Yaskawa INFORM job: X2_101(P)(125,-90)2.JBI

/JOB
//NAME X2_101(P)(125,-90)2
//POS
///NPOS 301,301,301,21,0,0
///TOOL 0
///POSTYPE PULSE
///PULSE
C00000=15474,202180,164610,0,0,38
C00001=2027,202198,164679,0,0,38
C00002=24736,215365,219614,34446,41710,-28276
C00003=32352,212431,219590,43411,47182,-30672
C00004=90146,188560,202920,30112,59119,-18336
C00005=118933,140461,218744,27304,53624,2807
C00006=105210,138110,229383,15554,54535,5056
C00007=120292,133807,224829,20615,58147,10246
C00008=120593,126537,218642,20775,58190,10295
C00009=120714,122004,214268,20769,58520,10378
C00010=120712,120035,212036,20692,58860,10445
C00011=120706,120595,212633,20705,58786,10429
C00012=120711,120851,214586,20937,57781,10229
C00013=120706,120595,212633,20705,58786,10429
C00014=120282,131035,221795,20517,58565,10327
C00015=120212,122631,223677,-19824,46644,-20033
C00016=120556,114962,216653,-19506,47024,-20076
C00017=120695,110312,211910,-19265,47534,-20168
C00018=120692,108202,209411,-19133,47963,-20258
C00019=120705,108724,209976,-19149,47889,-20241
C00020=120711,108700,211606,-19450,46928,-20036
C00021=120705,108724,209976,-19149,47889,-20241
C00022=120221,119783,220398,-19646,47168,-20147
C00023=120925,149751,244690,-34380,46703,-25518
C00024=121373,166523,227022,-36141,61926,-29055
C00025=120913,160748,223481,-36594,61174,-28897
C00026=120724,157112,220738,-36737,60983,-28874
C00027=120723,155199,218883,-36687,61111,-28923
C00028=120726,155677,219330,-36695,61088,-28913
C00029=120730,156730,222096,-37075,60150,-28553
C00030=120726,155677,219330,-36695,61088,-28913
C00031=121373,163920,224609,-36096,62046,-29099
C00032=120406,166637,227168,32311,57445,33728
C00033=120634,160817,223613,32676,56712,33541
C00034=120726,157198,220899,32780,56532,33504
C00035=120724,155250,219012,32723,56668,33550
C00036=120724,155690,219346,32716,56686,33555
C00037=120728,156742,222112,33132,55702,33215
C00038=120724,155690,219346,32716,56686,33555
C00039=120404,163997,224646,32246,57611,33783
C00040=133985,188744,240463,29202,55916,39414
C00041=133634,187862,227777,4842,42432,-77424
C00042=133983,183120,225880,4948,41153,-77374
C00043=134120,180360,224355,4989,40668,-77353
C00044=134108,178284,222610,4989,40676,-77358
C00045=134105,178637,222778,4981,40754,-77354
C00046=134286,180154,225906,5092,39605,-77360
C00047=134105,178637,222778,4981,40754,-77354
C00048=133615,185408,225690,4841,42456,-77429
C00049=121024,187697,227471,-25597,51015,-56291
C00050=120818,183050,225741,-26098,49773,-56012
C00051=120733,179873,223904,-26298,49302,-55905
C00052=120732,178247,222533,-26295,49309,-55908
C00053=120727,178630,222748,-26272,49366,-55926
C00054=120731,180176,225930,-26719,48320,-55616
C00055=120727,178630,222748,-26272,49366,-55926
C00056=121016,185268,225421,-25593,51025,-56296
C00057=120731,192327,238382,-525,21384,290
C00058=120720,184650,229554,-485,22872,268
C00059=120716,180491,225010,-470,23531,260
C00060=120714,178589,223412,-468,23537,258
C00061=120748,179412,224155,-490,23503,278
C00062=120744,177812,220907,-466,24679,265
C00063=120748,179412,224155,-490,23503,278
C00064=120764,190350,236905,-549,21277,311
C00065=148285,214402,237949,-4998,43525,10906
C00066=147844,206959,231028,-4889,43936,10712
C00067=147660,202909,227431,-4849,44060,10633
C00068=147643,201403,226399,-4857,43921,10635
C00069=147640,202124,226903,-4851,43981,10631
C00070=147319,200210,223567,-4711,45030,10450
C00071=147640,202124,226903,-4851,43981,10631
C00072=148254,212678,236902,-5015,43283,10908
C00073=144264,210294,243886,-8163,41086,13861
C00074=120755,180327,220298,-188,44229,164
C00075=120746,171881,211470,-184,45322,159
C00076=120742,168341,207661,-183,45847,157
C00077=120740,165439,205214,-182,45862,156
C00078=120719,166269,205935,-182,45844,148
C00079=120715,163797,201654,-178,47209,145
C00080=120719,166269,205935,-182,45844,148
C00081=120731,178408,218855,-188,44131,156
C00082=123087,177778,218562,-48004,45649,30777
C00083=121479,171146,210872,-47323,45938,29789
C00084=122530,166189,205678,-46713,46798,29742
C00085=122529,164979,204619,-46708,46819,29729
C00086=122529,165602,205165,-46719,46807,29736
C00087=122503,162924,200443,-45712,47877,29056
C00088=120838,166307,205861,-46999,46102,29364
C00089=120835,166361,205848,-46974,46126,29347
C00090=119861,166365,205849,-47111,45747,29113
C00091=120835,166361,205848,-46974,46126,29347
C00092=123074,175909,217070,-48037,45614,30794
C00093=121232,181774,235538,-27606,54021,27673
C00094=119095,158997,232657,-4189,63418,24156
C00095=116556,130755,220822,24696,63782,20050
C00096=116783,124225,216003,24912,63404,19994
C00097=116677,121428,213790,24861,63345,19966
C00098=124126,121440,213840,29408,62514,20795
C00099=124377,124183,215942,29533,62587,20852
C00100=123965,130725,220810,29194,62957,20896
C00101=125440,119589,219417,-31168,54029,-25826
C00102=124101,112544,213722,-32040,53801,-25914
C00103=124461,109637,211291,-31816,53838,-25883
C00104=115994,109663,211221,-37050,53005,-26653
C00105=116510,112581,213754,-36756,53014,-26588
C00106=116995,119639,219557,-36430,53113,-26564
C00107=126218,162099,239521,-28020,56999,-39411
C00108=123870,163328,223290,-28334,68014,-35019
C00109=122959,158598,221396,-29010,66719,-34890
C00110=123282,156546,220319,-28934,66438,-34739
C00111=117771,156561,220306,-31571,65347,-35721
C00112=117971,158636,221439,-31392,65705,-35782
C00113=118266,163418,223444,-30986,66822,-36040
C00114=120221,175834,229084,-3119,74575,4073
C00115=117582,163423,223451,27209,71262,31154
C00116=118328,158681,221539,27776,69997,31012
C00117=117739,156666,220543,27546,69730,30813
C00118=123312,156620,220547,30338,68636,31789
C00119=123482,158608,221419,30352,69024,31932
C00120=123188,163395,223433,29990,70147,32175
C00121=120067,178947,233192,25549,53044,55885
C00122=131070,185470,225867,7170,52227,-79323
C00123=131461,181907,225606,7389,50545,-79327
C00124=131646,180388,225354,7481,49912,-79321
C00125=136525,178881,222542,8029,50535,-77794
C00126=136445,180280,222598,7943,51220,-77765
C00127=135980,183829,222908,7713,52870,-77778
C00128=123522,184426,223985,-22802,61524,-57116
C00129=122967,181022,223967,-23325,59808,-56905
C00130=123040,179639,223960,-23465,59173,-56741
C00131=118101,179627,223904,-24803,58204,-57968
C00132=118290,181075,224034,-24590,58847,-58069
C00133=118546,184530,224142,-24121,60464,-58371
C00134=135828,184930,231784,3696,26075,2718
C00135=135741,176900,222633,3545,27580,2769
C00136=135898,173119,218034,3382,28468,2893
C00137=151866,161969,197943,-2562,35069,10366
C00138=151979,166024,202940,-2665,34080,10452
C00139=152363,175123,213641,-2941,32183,10704
C00140=121934,189549,236157,-2154,24440,9441
C00141=141176,183237,223578,-35123,36438,8037
C00142=140565,175008,214184,-33918,37549,7179
C00143=140340,171969,210603,-33443,38021,6842
C00144=125498,176939,219607,-33926,31237,2854
C00145=136257,146426,180013,-49389,59576,12695
C00146=136821,149913,184454,-49678,59198,13186
C00147=138256,158734,195155,-50257,58467,14304
C00148=90442,188267,218593,-20520,46484,-16259
C00149=38815,226894,234079,7619,30475,-17807
C00150=2027,202198,164679,0,0,38
C00151=15474,202180,164610,0,0,38
C00152=15474,202180,164610,0,0,38
C00153=15474,202180,164610,0,0,38
C00154=3643,-76224,-106676,19950,71810,76872
C00155=-17977,54134,16993,-10551,74333,28306
C00156=-37324,121541,115737,-14047,52289,7724
C00157=-48165,192898,197715,-15732,40765,-3970
C00158=-58614,195716,224396,-17895,28031,-14924
C00159=-138322,143321,229105,-42804,47301,-20408
C00160=-140817,146158,237227,-45779,45351,-19330
C00161=-147159,125749,218226,-45329,49662,-21330
C00162=-147437,121228,213779,-45242,49912,-21531
C00163=-147412,119200,211479,-45009,50185,-21684
C00164=-147407,119721,212016,-45043,50140,-21657
C00165=-147931,119949,213841,-45946,49334,-21289
C00166=-147407,119721,212016,-45043,50140,-21657
C00167=-146392,130285,221614,-44743,49966,-21354
C00168=-146532,144143,225646,4227,57465,17778
C00169=-147178,137204,219990,3902,57394,17672
C00170=-147427,133024,216151,3767,57613,17639
C00171=-147404,130928,213882,3765,57930,17654
C00172=-147409,131440,214347,3763,57908,17652
C00173=-147876,131929,216457,3567,56871,17542
C00174=-147409,131440,214347,3763,57908,17652
C00175=-146502,154568,235407,4272,56817,17758
C00176=-99845,140323,234668,41114,43975,29200
C00177=-130588,156406,235029,35449,55402,24493
C00178=-147611,165369,225951,24300,67303,24402
C00179=-147499,159686,222616,24499,66491,24247
C00180=-147440,155964,219836,24563,66297,24218
C00181=-147421,154162,218086,24545,66432,24252
C00182=-147416,154709,218664,24561,66363,24237
C00183=-147807,155692,221265,24569,65426,23941
C00184=-147416,154709,218664,24561,66363,24237
C00185=-147574,162825,223650,24300,67397,24430
C00186=-120351,165667,226538,-30553,61026,-29699
C00187=-120572,159826,222941,-30869,60298,-29533
C00188=-120662,156191,220198,-30959,60125,-29502
C00189=-120661,154235,218293,-30911,60269,-29546
C00190=-120662,154654,218578,-30900,60303,-29557
C00191=-120660,155573,221272,-31248,59284,-29233
C00192=-120662,154654,218578,-30900,60303,-29557
C00193=-120351,162993,223944,-30493,61219,-29757
C00194=-106019,170897,239329,-29591,39413,-48114
C00195=-120349,165701,226589,-30025,41462,-53269
C00196=-120571,159856,222988,-30524,40733,-53054
C00197=-120660,156245,220264,-30650,40558,-53013
C00198=-120659,154264,218337,-30550,40705,-53072
C00199=-120657,154705,218714,-30553,40700,-53069
C00200=-120657,155527,221042,-31160,39828,-52703
C00201=-120657,154705,218714,-30553,40700,-53069
C00202=-120346,163050,224086,-29924,41618,-53328
C00203=-121003,165681,226549,30422,41392,53375
C00204=-120764,159836,222944,30930,40664,53161
C00205=-120666,156628,220610,31078,40460,53111
C00206=-120665,154243,218290,30958,40635,53182
C00207=-120651,154718,218742,30981,40602,53173
C00208=-120645,155770,221512,31697,39599,52755
C00209=-120651,154718,218742,30981,40602,53173
C00210=-120988,163064,224120,30339,41520,53430
C00211=-145273,180969,224600,13907,25635,-13338
C00212=-150975,169052,202561,-14336,33678,-6171
C00213=-152120,157871,187736,-12805,36812,-7299
C00214=-151822,150501,178835,-12433,38503,-7437
C00215=-151822,147953,176273,-12361,38765,-7478
C00216=-151822,149084,177415,-12394,38645,-7460
C00217=-151589,146591,173415,-12167,39831,-7535
C00218=-151919,152197,181098,-12541,37982,-7398
C00219=-152280,169114,198720,-13043,35835,-7206
C00220=-158898,171274,210982,-44327,26584,1788
C00221=-158473,166641,205336,-42970,27544,1214
C00222=-157744,151580,188391,-39934,29853,-149
C00223=-157744,148965,185817,-39669,30040,-287
C00224=-157744,150293,187130,-39808,29943,-216
C00225=-157372,147876,183051,-38565,31072,-770
C00226=-157636,151887,188203,-39669,30105,-261
C00227=-158813,181767,219065,-43782,26920,1533
C00228=-129261,210513,245515,5534,45622,-8457
C00229=-125085,198862,239535,25777,46081,-13421
C00230=-119299,188173,224850,24885,48032,-10780
C00231=-120885,182304,217176,24168,49943,-10840
C00232=-120885,180234,215583,24199,49865,-10857
C00233=-120885,180747,215981,24191,49883,-10853
C00234=-120884,178818,212615,23832,50874,-10599
C00235=-120886,180612,215743,24164,49954,-10836
C00236=-120886,189219,222159,24004,50389,-10723
C00237=-108287,189347,219965,24064,48852,-6477
C00238=-108287,184786,216642,24169,48578,-6550
C00239=-108287,180112,213087,24246,48382,-6602
C00240=-108287,177544,211068,24278,48311,-6618
C00241=-108287,178306,211671,24271,48329,-6612
C00242=-108405,176503,208569,23922,49256,-6410
C00243=-108249,178868,212644,24384,48037,-6676
C00244=-121452,188951,222489,24083,50199,-10971
C00245=-121452,188951,222489,24083,50199,-10971
C00246=-122116,184054,218869,24132,50081,-11240
C00247=-122262,178348,212240,23732,51169,-11010
C00248=-108771,176193,208579,23747,49083,-6567
C00249=-111092,174695,211589,36295,46390,-11684
C00250=-112169,180872,218864,36952,45675,-12470
C00251=-113202,195859,242327,41337,40702,-15530
C00252=-130749,165712,222917,10388,27694,-8279
C00253=-152425,178401,240789,-26989,10054,1286
C00254=-149111,168631,221120,-26779,26556,407
C00255=-148536,165202,217049,-26272,27343,326
C00256=-159853,153774,193335,-13592,36205,-8842
C00257=-158113,149758,193299,-37101,31198,-1306
C00258=-158618,158017,203094,-38867,29614,-530
C00259=-160401,183295,230590,-43445,26035,1284
C00260=-117887,183372,223265,-22549,61468,-57164
C00261=-118052,179927,223173,-22955,59851,-56864
C00262=-118699,178546,222858,-23249,59248,-56921
C00263=-123672,178493,222758,-24591,58283,-58163
C00264=-123113,179961,223261,-24333,58805,-58120
C00265=-122866,183435,223403,-23872,60412,-58418
C00266=-123473,183399,223341,22943,61343,57288
C00267=-123290,179951,223242,23362,59727,56988
C00268=-123487,178672,223340,23471,59103,56791
C00269=-118424,178788,223621,24887,57983,58016
C00270=-118228,179938,223194,24724,58720,58254
C00271=-118494,183412,223341,24252,60324,58552
C00272=-131011,176479,228164,31225,71276,43628
C00273=-123827,162412,222773,27424,71320,31095
C00274=-123627,157628,220768,27711,70190,30861
C00275=-124009,155619,219621,27570,69971,30722
C00276=-118332,155649,219817,30457,68786,31689
C00277=-117906,157627,220734,30586,69092,31875
C00278=-118212,162433,222788,30219,70202,32114
C00279=-117529,162374,222654,-26899,71438,-31030
C00280=-117708,157592,220653,-27171,70307,-30797
C00281=-118564,155615,219745,-27674,69741,-30848
C00282=-124047,155559,219614,-30429,68730,-31821
C00283=-123427,157610,220727,-30053,69177,-31802
C00284=-123142,162415,222776,-29701,70290,-32041
C00285=-132073,148583,237547,-34621,60846,-21391
C00286=-129975,141241,222454,-31403,66136,-22661
C00287=-130468,135202,218431,-31833,65522,-22562
C00288=-131729,132640,216434,-32594,65253,-22701
C00289=-138385,131644,213865,-36199,65039,-23836
C00290=-137184,134500,216293,-35511,65228,-23678
C00291=-136557,140559,220416,-35003,65813,-23762
C00292=-150189,140118,219078,9123,71574,17400
C00293=-150541,134122,215115,8948,70956,17299
C00294=-151485,131353,212608,8387,71119,17166
C00295=-145176,132679,216974,12237,68813,17910
C00296=-144130,135523,219427,12862,68701,18051
C00297=-143910,141531,223338,12937,69351,18155
C00298=-134795,161184,236321,9699,64146,14551
C00299=-58614,195716,224396,-17895,28031,-14924
C00300=15474,202180,164610,0,0,38
BC00000=0,675528,1075229
BC00001=0,1249520,1075229
BC00002=20074,1273230,1075229
BC00003=22843,1276500,1075229
BC00004=181219,1349640,881743
BC00005=259614,1271622,997019
BC00006=263455,1253369,961473
BC00007=299365,1262893,899090
BC00008=299365,1262893,899090
BC00009=299365,1262893,899090
BC00010=299365,1262893,899090
BC00011=299365,1262893,899090
BC00012=299365,1262893,899090
BC00013=299365,1262893,899090
BC00014=299365,1262893,899090
BC00015=317385,1250080,966851
BC00016=317385,1250080,966851
BC00017=317385,1250080,966851
BC00018=317385,1250080,966851
BC00019=317385,1250080,966851
BC00020=317385,1250080,966851
BC00021=317385,1250080,966851
BC00022=317385,1250080,966851
BC00023=333821,1266832,919202
BC00024=286205,1304114,811613
BC00025=286205,1304114,811613
BC00026=286205,1304114,811613
BC00027=286205,1304114,811613
BC00028=286205,1304114,811613
BC00029=286205,1304114,811613
BC00030=286205,1304114,811613
BC00031=286205,1304114,811613
BC00032=312946,1307861,830398
BC00033=312946,1307861,830398
BC00034=312946,1307861,830398
BC00035=312946,1307861,830398
BC00036=312946,1307861,830398
BC00037=312946,1307861,830398
BC00038=312946,1307861,830398
BC00039=312946,1307861,830398
BC00040=309388,1296619,799441
BC00041=318547,1318060,813250
BC00042=318547,1318060,813250
BC00043=318547,1318060,813250
BC00044=318547,1318060,813250
BC00045=318547,1318060,813250
BC00046=318547,1318060,813250
BC00047=318547,1318060,813250
BC00048=318547,1318060,813250
BC00049=305027,1313604,795360
BC00050=305027,1313604,795360
BC00051=305027,1313604,795360
BC00052=305027,1313604,795360
BC00053=305027,1313604,795360
BC00054=305027,1313604,795360
BC00055=305027,1313604,795360
BC00056=305027,1313604,795360
BC00057=324377,1352422,788984
BC00058=324377,1352422,788984
BC00059=324377,1352422,788984
BC00060=324377,1352422,788984
BC00061=324377,1352422,788984
BC00062=324377,1352422,788984
BC00063=324377,1352422,788984
BC00064=324377,1352422,788984
BC00065=364692,1338716,661668
BC00066=364692,1338716,661668
BC00067=364692,1338716,661668
BC00068=364692,1338716,661668
BC00069=364692,1338716,661668
BC00070=364692,1338716,661668
BC00071=364692,1338716,661668
BC00072=364692,1338716,661668
BC00073=369598,1321086,746352
BC00074=329275,1315048,881081
BC00075=329275,1315048,881081
BC00076=329275,1315048,881081
BC00077=329275,1315048,881081
BC00078=329275,1315048,881081
BC00079=329275,1315048,881081
BC00080=329275,1315048,881081
BC00081=329275,1315048,881081
BC00082=314852,1330108,807446
BC00083=314852,1330108,807446
BC00084=314853,1330108,807444
BC00085=314853,1330108,807443
BC00086=314853,1330108,807443
BC00087=314853,1330108,807443
BC00088=314852,1330108,807446
BC00089=314852,1330108,807446
BC00090=314852,1330108,807446
BC00091=314852,1330108,807446
BC00092=314852,1330108,807446
BC00093=313257,1310637,824311
BC00094=311421,1288215,843732
BC00095=309154,1260535,867707
BC00096=309154,1260535,867707
BC00097=309154,1260535,867707
BC00098=309154,1260535,867707
BC00099=309154,1260535,867707
BC00100=309154,1260535,867707
BC00101=294407,1249819,928832
BC00102=294407,1249819,928832
BC00103=294407,1249819,928832
BC00104=294407,1249819,928832
BC00105=294407,1249819,928832
BC00106=294407,1249819,928832
BC00107=314801,1292959,892910
BC00108=293885,1292722,795471
BC00109=293885,1292722,795471
BC00110=293885,1292722,795471
BC00111=293885,1292722,795471
BC00112=293885,1292722,795471
BC00113=293885,1292722,795471
BC00114=299435,1291649,781795
BC00115=313202,1288383,786633
BC00116=313202,1288383,786633
BC00117=313202,1288383,786633
BC00118=313201,1288384,786631
BC00119=313202,1288383,786633
BC00120=313202,1288383,786633
BC00121=311248,1293583,920117
BC00122=320223,1301498,798955
BC00123=320223,1301498,798955
BC00124=320223,1301498,798955
BC00125=320223,1301498,798955
BC00126=320223,1301498,798955
BC00127=320223,1301498,798955
BC00128=303809,1297500,774731
BC00129=303809,1297500,774731
BC00130=303809,1297500,774731
BC00131=303809,1297500,774731
BC00132=303809,1297500,774731
BC00133=303809,1297500,774731
BC00134=382985,1337291,817528
BC00135=382985,1337291,817528
BC00136=382985,1337291,817528
BC00137=382985,1337291,817528
BC00138=382985,1337291,817528
BC00139=382985,1337291,817528
BC00140=326395,1340304,844891
BC00141=362940,1334773,820893
BC00142=362940,1334773,820893
BC00143=362940,1334773,820893
BC00144=362940,1334773,820893
BC00145=362940,1334773,820893
BC00146=362940,1334773,820893
BC00147=362940,1334773,820893
BC00148=199115,1355011,996382
BC00149=79950,1309724,1030230
BC00150=0,1249520,1075229
BC00151=0,675528,1075229
BC00152=0,675528,1075229
BC00153=0,675528,1075229
BC00154=199464,674570,1075173
BC00155=168150,723863,951549
BC00156=154085,663617,1001676
BC00157=146204,714236,1057448
BC00158=138607,763027,1056836
BC00159=343461,851890,923082
BC00160=347349,853577,920544
BC00161=364317,860937,909465
BC00162=364317,860937,909465
BC00163=364317,860937,909465
BC00164=364317,860937,909465
BC00165=364317,860937,909465
BC00166=364317,860937,909465
BC00167=364317,860937,909465
BC00168=379202,846237,874129
BC00169=379202,846237,874129
BC00170=379202,846237,874129
BC00171=379202,846237,874129
BC00172=379202,846237,874129
BC00173=379202,846237,874129
BC00174=379202,846237,874129
BC00175=379202,846237,874129
BC00176=267497,855485,958441
BC00177=320924,819371,961652
BC00178=359813,832026,812779
BC00179=359813,832026,812779
BC00180=359813,832026,812779
BC00181=359813,832026,812779
BC00182=359813,832026,812779
BC00183=359813,832026,812779
BC00184=359813,832026,812779
BC00185=359813,832026,812779
BC00186=313650,822927,822655
BC00187=313650,822927,822655
BC00188=313650,822927,822655
BC00189=313650,822927,822655
BC00190=313650,822927,822655
BC00191=313650,822927,822655
BC00192=313650,822927,822655
BC00193=313650,822927,822655
BC00194=268540,837164,928608
BC00195=303309,837622,929453
BC00196=303309,837622,929453
BC00197=303309,837622,929453
BC00198=303309,837622,929453
BC00199=303309,837622,929453
BC00200=303309,837622,929453
BC00201=303309,837622,929453
BC00202=303309,837622,929453
BC00203=306476,837214,930249
BC00204=306476,837214,930249
BC00205=306476,837214,930249
BC00206=306476,837214,930249
BC00207=306476,837214,930249
BC00208=306476,837214,930249
BC00209=306476,837214,930249
BC00210=306476,837214,930249
BC00211=398174,775712,811563
BC00212=398174,775712,811563
BC00213=398174,775712,811563
BC00214=398174,775712,811563
BC00215=398174,775712,811563
BC00216=398174,775712,811563
BC00217=398174,775712,811563
BC00218=398174,775712,811563
BC00219=398174,775712,811563
BC00220=398174,793888,811563
BC00221=398174,793888,811563
BC00222=398174,793888,811563
BC00223=398174,793888,811563
BC00224=398174,793888,811563
BC00225=398174,793888,811563
BC00226=398174,793888,811563
BC00227=398174,793888,811563
BC00228=296475,807012,791430
BC00229=296475,807012,791430
BC00230=296475,807012,791430
BC00231=296475,807012,791430
BC00232=296475,807012,791430
BC00233=296475,807012,791430
BC00234=296475,807012,791430
BC00235=296475,807012,791430
BC00236=296475,807012,791430
BC00237=296475,807012,791430
BC00238=296475,807012,791430
BC00239=296475,807012,791430
BC00240=296475,807012,791430
BC00241=296475,807012,791430
BC00242=296475,807012,791430
BC00243=296475,807012,791430
BC00244=296475,807012,791430
BC00245=296475,807012,791430
BC00246=296475,807012,791430
BC00247=296476,807010,791427
BC00248=296786,806946,791584
BC00249=296786,806946,791584
BC00250=296786,806946,791584
BC00251=296786,806946,791584
BC00252=343473,807454,949850
BC00253=383324,814067,855911
BC00254=383324,814067,855911
BC00255=383324,814067,855911
BC00256=383324,814066,855908
BC00257=383324,814067,855911
BC00258=383324,814067,855911
BC00259=383324,814067,855911
BC00260=304526,826961,775443
BC00261=304526,826961,775443
BC00262=304526,826961,775443
BC00263=304526,826961,775443
BC00264=304526,826961,775443
BC00265=304526,826961,775443
BC00266=305115,826537,776504
BC00267=305115,826537,776504
BC00268=305115,826537,776504
BC00269=305115,826537,776504
BC00270=305115,826537,776504
BC00271=305115,826537,776504
BC00272=317689,831131,771467
BC00273=295274,836215,786981
BC00274=295274,836215,786981
BC00275=295274,836215,786981
BC00276=295274,836215,786981
BC00277=295274,836215,786981
BC00278=295274,836215,786981
BC00279=313970,836931,785826
BC00280=313970,836931,785826
BC00281=313970,836931,785826
BC00282=313970,836931,785826
BC00283=313970,836931,785826
BC00284=313970,836931,785826
BC00285=304168,872987,860177
BC00286=340834,848874,817062
BC00287=340834,848874,817062
BC00288=340834,848874,817062
BC00289=340834,848874,817062
BC00290=340834,848874,817062
BC00291=340834,848874,817062
BC00292=360407,856018,818040
BC00293=360407,856018,818040
BC00294=360407,856018,818040
BC00295=360407,856018,818040
BC00296=360407,856018,818040
BC00297=360407,856018,818040
BC00298=336693,846075,843572
BC00299=138607,763027,1056836
BC00300=0,675528,1075229
EC00000=1108551,-556475
EC00001=1108551,-556475
EC00002=1108551,-556475
EC00003=1108551,-556475
EC00004=1108551,-556475
EC00005=1108551,-556475
EC00006=1108551,-556475
EC00007=1108551,-556475
EC00008=1108551,-556475
EC00009=1108551,-556475
EC00010=1108551,-556475
EC00011=1108551,-556475
EC00012=1108551,-556475
EC00013=1108551,-556475
EC00014=1108551,-556475
EC00015=1108551,-556475
EC00016=1108551,-556475
EC00017=1108551,-556475
EC00018=1108551,-556475
EC00019=1108551,-556475
EC00020=1108551,-556475
EC00021=1108551,-556475
EC00022=1108551,-556475
EC00023=1108551,-556475
EC00024=1108551,-556475
EC00025=1108551,-556475
EC00026=1108551,-556475
EC00027=1108551,-556475
EC00028=1108551,-556475
EC00029=1108551,-556475
EC00030=1108551,-556475
EC00031=1108551,-556475
EC00032=1108551,-556475
EC00033=1108551,-556475
EC00034=1108551,-556475
EC00035=1108551,-556475
EC00036=1108551,-556475
EC00037=1108551,-556475
EC00038=1108551,-556475
EC00039=1108551,-556475
EC00040=1108551,-556475
EC00041=1108551,-556475
EC00042=1108551,-556475
EC00043=1108551,-556475
EC00044=1108551,-556475
EC00045=1108551,-556475
EC00046=1108551,-556475
EC00047=1108551,-556475
EC00048=1108551,-556475
EC00049=1108551,-556475
EC00050=1108551,-556475
EC00051=1108551,-556475
EC00052=1108551,-556475
EC00053=1108551,-556475
EC00054=1108551,-556475
EC00055=1108551,-556475
EC00056=1108551,-556475
EC00057=1108551,-556475
EC00058=1108551,-556475
EC00059=1108551,-556475
EC00060=1108551,-556475
EC00061=1108551,-556475
EC00062=1108551,-556475
EC00063=1108551,-556475
EC00064=1108551,-556475
EC00065=1108551,-556475
EC00066=1108551,-556475
EC00067=1108551,-556475
EC00068=1108551,-556475
EC00069=1108551,-556475
EC00070=1108551,-556475
EC00071=1108551,-556475
EC00072=1108551,-556475
EC00073=1108551,-556475
EC00074=1108551,-556475
EC00075=1108551,-556475
EC00076=1108551,-556475
EC00077=1108551,-556475
EC00078=1108551,-556475
EC00079=1108551,-556475
EC00080=1108551,-556475
EC00081=1108551,-556475
EC00082=1108551,-556475
EC00083=1108551,-556475
EC00084=1108551,-556475
EC00085=1108550,-556475
EC00086=1108550,-556475
EC00087=1108550,-556475
EC00088=1108551,-556475
EC00089=1108551,-556475
EC00090=1108551,-556475
EC00091=1108551,-556475
EC00092=1108551,-556475
EC00093=1108551,-556475
EC00094=1108551,-556475
EC00095=1108551,-556475
EC00096=1108551,-556475
EC00097=1108551,-556475
EC00098=1108551,-556475
EC00099=1108551,-556475
EC00100=1108551,-556475
EC00101=1108551,-556475
EC00102=1108551,-556475
EC00103=1108551,-556475
EC00104=1108551,-556475
EC00105=1108551,-556475
EC00106=1108551,-556475
EC00107=1108551,-556475
EC00108=1108551,-556475
EC00109=1108551,-556475
EC00110=1108551,-556475
EC00111=1108551,-556475
EC00112=1108551,-556475
EC00113=1108551,-556475
EC00114=1108551,-556475
EC00115=1108551,-556475
EC00116=1108551,-556475
EC00117=1108551,-556475
EC00118=1108550,-556474
EC00119=1108551,-556475
EC00120=1108551,-556475
EC00121=1108551,-556475
EC00122=1108551,-556475
EC00123=1108551,-556475
EC00124=1108551,-556475
EC00125=1108551,-556475
EC00126=1108551,-556475
EC00127=1108551,-556475
EC00128=1108551,-556475
EC00129=1108551,-556475
EC00130=1108551,-556475
EC00131=1108551,-556475
EC00132=1108551,-556475
EC00133=1108551,-556475
EC00134=1108551,-556475
EC00135=1108551,-556475
EC00136=1108551,-556475
EC00137=1108551,-556475
EC00138=1108551,-556475
EC00139=1108551,-556475
EC00140=1108551,-556475
EC00141=1108551,-556475
EC00142=1108551,-556475
EC00143=1108551,-556475
EC00144=1108551,-556475
EC00145=1108551,-556475
EC00146=1108551,-556475
EC00147=1108551,-556475
EC00148=1108551,-556475
EC00149=1108551,-556475
EC00150=1108551,-556475
EC00151=1108551,-556475
EC00152=266052,-556475
EC00153=-266052,556475
EC00154=-1108551,556475
EC00155=-1108551,556475
EC00156=-1108551,556475
EC00157=-1108551,556475
EC00158=-1108551,556475
EC00159=-1108551,556475
EC00160=-1108551,556475
EC00161=-1108551,556475
EC00162=-1108551,556475
EC00163=-1108551,556475
EC00164=-1108551,556475
EC00165=-1108551,556475
EC00166=-1108551,556475
EC00167=-1108551,556475
EC00168=-1108551,556475
EC00169=-1108551,556475
EC00170=-1108551,556475
EC00171=-1108551,556475
EC00172=-1108551,556475
EC00173=-1108551,556475
EC00174=-1108551,556475
EC00175=-1108551,556475
EC00176=-1108551,556475
EC00177=-1108551,556475
EC00178=-1108551,556475
EC00179=-1108551,556475
EC00180=-1108551,556475
EC00181=-1108551,556475
EC00182=-1108551,556475
EC00183=-1108551,556475
EC00184=-1108551,556475
EC00185=-1108551,556475
EC00186=-1108551,556475
EC00187=-1108551,556475
EC00188=-1108551,556475
EC00189=-1108551,556475
EC00190=-1108551,556475
EC00191=-1108551,556475
EC00192=-1108551,556475
EC00193=-1108551,556475
EC00194=-1108551,556475
EC00195=-1108551,556475
EC00196=-1108551,556475
EC00197=-1108551,556475
EC00198=-1108551,556475
EC00199=-1108551,556475
EC00200=-1108551,556475
EC00201=-1108551,556475
EC00202=-1108551,556475
EC00203=-1108551,556475
EC00204=-1108551,556475
EC00205=-1108551,556475
EC00206=-1108551,556475
EC00207=-1108551,556475
EC00208=-1108551,556475
EC00209=-1108551,556475
EC00210=-1108551,556475
EC00211=-1108551,556475
EC00212=-1108551,556475
EC00213=-1108551,556475
EC00214=-1108551,556475
EC00215=-1108551,556475
EC00216=-1108551,556475
EC00217=-1108551,556475
EC00218=-1108551,556475
EC00219=-1108551,556475
EC00220=-1108551,556475
EC00221=-1108551,556475
EC00222=-1108551,556475
EC00223=-1108551,556475
EC00224=-1108551,556475
EC00225=-1108551,556475
EC00226=-1108551,556475
EC00227=-1108551,556475
EC00228=-1108551,556475
EC00229=-1108551,556475
EC00230=-1108551,556475
EC00231=-1108551,556475
EC00232=-1108551,556475
EC00233=-1108551,556475
EC00234=-1108551,556475
EC00235=-1108551,556475
EC00236=-1108551,556475
EC00237=-1108551,556475
EC00238=-1108551,556475
EC00239=-1108551,556475
EC00240=-1108551,556475
EC00241=-1108551,556475
EC00242=-1108551,556475
EC00243=-1108551,556475
EC00244=-1108551,556475
EC00245=-1108551,556475
EC00246=-1108551,556475
EC00247=-1108549,556475
EC00248=-1108549,556475
EC00249=-1108549,556475
EC00250=-1108549,556475
EC00251=-1108549,556475
EC00252=-1108551,556475
EC00253=-1108551,556475
EC00254=-1108551,556475
EC00255=-1108551,556475
EC00256=-1108550,556475
EC00257=-1108551,556475
EC00258=-1108551,556475
EC00259=-1108551,556475
EC00260=-1108551,556475
EC00261=-1108551,556475
EC00262=-1108551,556475
EC00263=-1108551,556475
EC00264=-1108551,556475
EC00265=-1108551,556475
EC00266=-1108551,556475
EC00267=-1108551,556475
EC00268=-1108551,556475
EC00269=-1108551,556475
EC00270=-1108551,556475
EC00271=-1108551,556475
EC00272=-1108551,556475
EC00273=-1108551,556475
EC00274=-1108551,556475
EC00275=-1108551,556475
EC00276=-1108551,556475
EC00277=-1108551,556475
EC00278=-1108551,556475
EC00279=-1108551,556475
EC00280=-1108551,556475
EC00281=-1108551,556475
EC00282=-1108551,556475
EC00283=-1108551,556475
EC00284=-1108551,556475
EC00285=-1108551,556475
EC00286=-1108551,556475
EC00287=-1108551,556475
EC00288=-1108551,556475
EC00289=-1108551,556475
EC00290=-1108551,556475
EC00291=-1108551,556475
EC00292=-1108551,556475
EC00293=-1108551,556475
EC00294=-1108551,556475
EC00295=-1108551,556475
EC00296=-1108551,556475
EC00297=-1108551,556475
EC00298=-1108551,556475
EC00299=-1108551,556475
EC00300=-1108551,556475
///POSTYPE BASE
///RECTAN
///RCONF 0,0,0,0,0,0,0,0,0,0,0,0,0,0,0,0,0,0,0,0,0,0,0,0
P00006=0.222,-3.123,-1.508,0.0000,0.0000,0.0000
P00021=-0.225,-6.128,-0.405,0.0000,0.0000,0.0000
P00022=0.222,-3.123,-1.508,0.0000,0.0000,0.0000
P00024=0.145,-0.552,1.326,0.0000,0.0000,0.0000
P00025=-2.003,0.006,0.728,0.0000,0.0000,0.0000
P00027=-0.746,0.015,-9.096,0.0000,0.0000,0.0000
P00028=-2.237,-0.018,-7.702,0.0000,0.0000,0.0000
P00030=5.926,-4.294,-1.390,0.0000,0.0000,0.0000
P00031=1.853,-0.001,-1.549,0.0000,0.0000,0.0000
P00032=1.957,0.503,-7.217,0.0000,0.0000,0.0000
///RCONF 0,0,0,0,1,0,0,0,0,0,0,0,0,0,0,0,0,0,0,0,0,0,0,0
P00033=-0.123,0.612,-5.012,0.0000,0.0000,0.0000
///RCONF 0,0,0,0,0,0,0,0,0,0,0,0,0,0,0,0,0,0,0,0,0,0,0,0
P00041=0.192,3.924,0.305,0.0000,0.0000,0.0000
P00042=-0.217,1.941,0.413,0.0000,0.0000,0.0000
P00044=0.687,-2.322,1.156,0.0000,0.0000,0.0000
P00045=-0.068,-0.810,1.603,0.0000,0.0000,0.0000
///RCONF 0,1,0,0,0,0,0,0,0,0,0,0,0,0,0,0,0,0,0,0,0,0,0,0
P00047=-0.011,1.737,-0.646,0.0000,0.0000,0.0000
///RCONF 0,0,0,0,0,0,0,0,0,0,0,0,0,0,0,0,0,0,0,0,0,0,0,0
P00048=2.411,0.025,-0.606,0.0000,0.0000,0.0000
P00050=4.296,-4.501,-0.826,0.0000,0.0000,0.0000
P00051=0.367,3.892,0.009,0.0000,0.0000,0.0000
P00052=0.088,2.832,-0.342,0.0000,0.0000,0.0000
P00053=0.134,6.594,0.107,0.0000,0.0000,0.0000
//INST
///DATE 2024/11/05 12:02
///ATTR SC,RW
///GROUP1 RB1,BS1
///GROUP2 ST1
NOP
'X2_101(P)(125,-90)2
'
MOVJ C00000 BC00000 VJ=100.00  +MOVJ EC00000 VJ=100.00
MOVJ C00001 BC00001 VJ=100.00  +MOVJ EC00001 VJ=100.00
'
MOVJ C00002 BC00002 VJ=100.00  +MOVJ EC00002 VJ=100.00
MOVJ C00003 BC00003 VJ=100.00  +MOVJ EC00003 VJ=100.00
MOVJ C00004 BC00004 VJ=100.00  +MOVJ EC00004 VJ=100.00
MOVJ C00005 BC00005 VJ=100.00  +MOVJ EC00005 VJ=100.00
MOVJ C00006 BC00006 VJ=100.00  +MOVJ EC00006 VJ=100.00
'Path S3411
SFTOF3D
MOVJ C00007 BC00007 VJ=100.00  +MOVJ EC00007 VJ=100.00
MOVL C00008 BC00008 V=800.0  +MOVJ EC00008 VJ=100.00
SMOVL C00009 BC00009 V=166.7  +MOVJ EC00009
SREFP 3 C00010 BC00010  +REFP EC00010
CALL JOB:SEARCH-R1-S13D
SET P021 P006
SFTON3D P021
SMOVL C00011 BC00011 V=166.7  +MOVJ EC00011
SREFP 3 C00012 BC00012  +REFP EC00012
CALL JOB:SEARCH-R1-S13D
SET P021 P006
SFTON3D P021
SMOVL C00013 BC00013 V=166.7  +MOVJ EC00013
MOVL C00014 BC00014 V=1000.0  +MOVJ EC00014 VJ=100.00
'EndPath S3411
'Path S3412
SFTOF3D
MOVJ C00015 BC00015 VJ=100.00  +MOVJ EC00015 VJ=100.00
MOVL C00016 BC00016 V=800.0  +MOVJ EC00016 VJ=100.00
SMOVL C00017 BC00017 V=166.7  +MOVJ EC00017
SREFP 3 C00018 BC00018  +REFP EC00018
CALL JOB:SEARCH-R1-S13D
SET P022 P006
SFTON3D P022
SMOVL C00019 BC00019 V=166.7  +MOVJ EC00019
SREFP 3 C00020 BC00020  +REFP EC00020
CALL JOB:SEARCH-R1-S13D
SET P022 P006
SFTON3D P022
SMOVL C00021 BC00021 V=166.7  +MOVJ EC00021
MOVL C00022 BC00022 V=1000.0  +MOVJ EC00022 VJ=100.00
'EndPath S3412
MOVJ C00023 BC00023 VJ=100.00  +MOVJ EC00023 VJ=100.00
'Path S3414
SFTOF3D
MOVJ C00024 BC00024 VJ=100.00  +MOVJ EC00024 VJ=100.00
MOVL C00025 BC00025 V=800.0  +MOVJ EC00025 VJ=100.00
SMOVL C00026 BC00026 V=166.7  +MOVJ EC00026
SREFP 3 C00027 BC00027  +REFP EC00027
CALL JOB:SEARCH-R1-S13D
SET P024 P006
SFTON3D P024
SMOVL C00028 BC00028 V=166.7  +MOVJ EC00028
SREFP 3 C00029 BC00029  +REFP EC00029
CALL JOB:SEARCH-R1-S13D
SET P024 P006
SFTON3D P024
SMOVL C00030 BC00030 V=166.7  +MOVJ EC00030
MOVL C00031 BC00031 V=1000.0  +MOVJ EC00031 VJ=100.00
'EndPath S3414
'Path S3415
SFTOF3D
MOVJ C00032 BC00032 VJ=100.00  +MOVJ EC00032 VJ=100.00
MOVL C00033 BC00033 V=800.0  +MOVJ EC00033 VJ=100.00
SMOVL C00034 BC00034 V=166.7  +MOVJ EC00034
SREFP 3 C00035 BC00035  +REFP EC00035
CALL JOB:SEARCH-R1-S13D
SET P025 P006
SFTON3D P025
SMOVL C00036 BC00036 V=166.7  +MOVJ EC00036
SREFP 3 C00037 BC00037  +REFP EC00037
CALL JOB:SEARCH-R1-S13D
SET P025 P006
SFTON3D P025
SMOVL C00038 BC00038 V=166.7  +MOVJ EC00038
MOVL C00039 BC00039 V=1000.0  +MOVJ EC00039 VJ=100.00
'EndPath S3415
MOVJ C00040 BC00040 VJ=100.00  +MOVJ EC00040 VJ=100.00
'Path S3417
SFTOF3D
MOVJ C00041 BC00041 VJ=100.00  +MOVJ EC00041 VJ=100.00
MOVL C00042 BC00042 V=800.0  +MOVJ EC00042 VJ=100.00
SMOVL C00043 BC00043 V=166.7  +MOVJ EC00043
SREFP 3 C00044 BC00044  +REFP EC00044
CALL JOB:SEARCH-R1-S13D
SET P027 P006
SFTON3D P027
SMOVL C00045 BC00045 V=166.7  +MOVJ EC00045
SREFP 3 C00046 BC00046  +REFP EC00046
CALL JOB:SEARCH-R1-S13D
SET P027 P006
SFTON3D P027
SMOVL C00047 BC00047 V=166.7  +MOVJ EC00047
MOVL C00048 BC00048 V=1000.0  +MOVJ EC00048 VJ=100.00
'EndPath S3417
'Path S3418
SFTOF3D
MOVJ C00049 BC00049 VJ=100.00  +MOVJ EC00049 VJ=100.00
MOVL C00050 BC00050 V=800.0  +MOVJ EC00050 VJ=100.00
SMOVL C00051 BC00051 V=166.7  +MOVJ EC00051
SREFP 3 C00052 BC00052  +REFP EC00052
CALL JOB:SEARCH-R1-S13D
SET P028 P006
SFTON3D P028
SMOVL C00053 BC00053 V=166.7  +MOVJ EC00053
SREFP 3 C00054 BC00054  +REFP EC00054
CALL JOB:SEARCH-R1-S13D
SET P028 P006
SFTON3D P028
SMOVL C00055 BC00055 V=166.7  +MOVJ EC00055
MOVL C00056 BC00056 V=1000.0  +MOVJ EC00056 VJ=100.00
'EndPath S3418
'Path S3420
SFTOF3D
MOVJ C00057 BC00057 VJ=100.00  +MOVJ EC00057 VJ=100.00
MOVL C00058 BC00058 V=800.0  +MOVJ EC00058 VJ=100.00
SMOVL C00059 BC00059 V=166.7  +MOVJ EC00059
SREFP 3 C00060 BC00060  +REFP EC00060
CALL JOB:SEARCH-R1-S13D
SET P030 P006
SFTON3D P030
SMOVL C00061 BC00061 V=166.7  +MOVJ EC00061
SREFP 3 C00062 BC00062  +REFP EC00062
CALL JOB:SEARCH-R1-S13D
SET P030 P006
SFTON3D P030
SMOVL C00063 BC00063 V=166.7  +MOVJ EC00063
MOVL C00064 BC00064 V=1000.0  +MOVJ EC00064 VJ=100.00
'EndPath S3420
'Path S3421
SFTOF3D
MOVJ C00065 BC00065 VJ=100.00  +MOVJ EC00065 VJ=100.00
MOVL C00066 BC00066 V=800.0  +MOVJ EC00066 VJ=100.00
SMOVL C00067 BC00067 V=166.7  +MOVJ EC00067
SREFP 3 C00068 BC00068  +REFP EC00068
CALL JOB:SEARCH-R1-S13D
SET P031 P006
SFTON3D P031
SMOVL C00069 BC00069 V=166.7  +MOVJ EC00069
SREFP 3 C00070 BC00070  +REFP EC00070
CALL JOB:SEARCH-R1-S13D
SET P031 P006
SFTON3D P031
SMOVL C00071 BC00071 V=166.7  +MOVJ EC00071
MOVL C00072 BC00072 V=1000.0  +MOVJ EC00072 VJ=100.00
'EndPath S3421
MOVJ C00073 BC00073 VJ=100.00  +MOVJ EC00073 VJ=100.00
'Path S3422
SFTOF3D
MOVJ C00074 BC00074 VJ=100.00  +MOVJ EC00074 VJ=100.00
MOVL C00075 BC00075 V=800.0  +MOVJ EC00075 VJ=100.00
SMOVL C00076 BC00076 V=166.7  +MOVJ EC00076
SREFP 3 C00077 BC00077  +REFP EC00077
CALL JOB:SEARCH-R1-S13D
SET P032 P006
SFTON3D P032
SMOVL C00078 BC00078 V=166.7  +MOVJ EC00078
SREFP 3 C00079 BC00079  +REFP EC00079
CALL JOB:SEARCH-R1-S13D
SET P032 P006
SFTON3D P032
SMOVL C00080 BC00080 V=166.7  +MOVJ EC00080
MOVL C00081 BC00081 V=1000.0  +MOVJ EC00081 VJ=100.00
'EndPath S3422
'Path S3423
SFTOF3D
MOVJ C00082 BC00082 VJ=100.00  +MOVJ EC00082 VJ=100.00
MOVL C00083 BC00083 V=800.0  +MOVJ EC00083 VJ=100.00
SMOVL C00084 BC00084 V=166.7  +MOVJ EC00084
SREFP 3 C00085 BC00085  +REFP EC00085
CALL JOB:SEARCH-R1-S13D
SET P033 P006
SFTON3D P033
SMOVL C00086 BC00086 V=166.7  +MOVJ EC00086
SREFP 3 C00087 BC00087  +REFP EC00087
CALL JOB:SEARCH-R1-S13D
SET P033 P006
SFTON3D P033
SMOVL C00088 BC00088 V=166.7  +MOVJ EC00088
SMOVL C00089 BC00089 V=166.7  +MOVJ EC00089
SREFP 3 C00090 BC00090  +REFP EC00090
CALL JOB:SEARCH-R1-S13D
SET P033 P006
SFTON3D P033
SMOVL C00091 BC00091 V=166.7  +MOVJ EC00091
MOVL C00092 BC00092 V=1000.0  +MOVJ EC00092 VJ=100.00
'EndPath S3423
MOVJ C00093 BC00093 VJ=100.00  +MOVJ EC00093 VJ=100.00
MOVJ C00094 BC00094 VJ=100.00  +MOVJ EC00094 VJ=100.00
'Path W3424
SFTOF3D
SFTON3D P021
MOVJ C00095 BC00095 VJ=100.00  +MOVJ EC00095 VJ=100.00
SMOVL C00096 BC00096 V=800.0  +MOVJ EC00096
SMOVL C00097 BC00097 V=150.0 PL=0  +MOVJ EC00097
MACRO1 MJ#(0) ARGF9
ARCON
SMOVL C00098 BC00098 V=11.7  +MOVJ EC00098
ARCOF
SMOVL C00099 BC00099 V=800.0  +MOVJ EC00099
SMOVL C00100 BC00100 V=1000.0  +MOVJ EC00100
SFTOF3D
'EndPath W3424
'Path W3425
SFTOF3D
SFTON3D P022
MOVJ C00101 BC00101 VJ=100.00  +MOVJ EC00101 VJ=100.00
SMOVL C00102 BC00102 V=800.0  +MOVJ EC00102
SMOVL C00103 BC00103 V=150.0 PL=0  +MOVJ EC00103
ARCON
SMOVL C00104 BC00104 V=11.7  +MOVJ EC00104
ARCOF
SMOVL C00105 BC00105 V=800.0  +MOVJ EC00105
SMOVL C00106 BC00106 V=1000.0  +MOVJ EC00106
SFTOF3D
'EndPath W3425
'
MOVJ C00107 BC00107 VJ=100.00  +MOVJ EC00107 VJ=100.00
'Path W3427
SFTOF3D
SFTON3D P024
MOVJ C00108 BC00108 VJ=100.00  +MOVJ EC00108 VJ=100.00
SMOVL C00109 BC00109 V=800.0  +MOVJ EC00109
SMOVL C00110 BC00110 V=150.0 PL=0  +MOVJ EC00110
ARCON
SMOVL C00111 BC00111 V=11.7  +MOVJ EC00111
ARCOF
SMOVL C00112 BC00112 V=800.0  +MOVJ EC00112
SMOVL C00113 BC00113 V=1000.0  +MOVJ EC00113
SFTOF3D
'EndPath W3427
MOVJ C00114 BC00114 VJ=100.00  +MOVJ EC00114 VJ=100.00
'Path W3428
SFTOF3D
SFTON3D P025
MOVJ C00115 BC00115 VJ=100.00  +MOVJ EC00115 VJ=100.00
SMOVL C00116 BC00116 V=800.0  +MOVJ EC00116
SMOVL C00117 BC00117 V=150.0 PL=0  +MOVJ EC00117
ARCON
SMOVL C00118 BC00118 V=11.7  +MOVJ EC00118
ARCOF
SMOVL C00119 BC00119 V=800.0  +MOVJ EC00119
SMOVL C00120 BC00120 V=1000.0  +MOVJ EC00120
SFTOF3D
'EndPath W3428
'
MOVJ C00121 BC00121 VJ=100.00  +MOVJ EC00121 VJ=100.00
'Path W3430
SFTOF3D
SFTON3D P027
MOVJ C00122 BC00122 VJ=100.00  +MOVJ EC00122 VJ=100.00
SMOVL C00123 BC00123 V=800.0  +MOVJ EC00123
SMOVL C00124 BC00124 V=150.0 PL=0  +MOVJ EC00124
ARCON
SMOVL C00125 BC00125 V=10.0  +MOVJ EC00125
ARCOF
SMOVL C00126 BC00126 V=800.0  +MOVJ EC00126
SMOVL C00127 BC00127 V=1000.0  +MOVJ EC00127
SFTOF3D
'EndPath W3430
'Path W3431
SFTOF3D
SFTON3D P028
MOVJ C00128 BC00128 VJ=100.00  +MOVJ EC00128 VJ=100.00
SMOVL C00129 BC00129 V=800.0  +MOVJ EC00129
SMOVL C00130 BC00130 V=150.0 PL=0  +MOVJ EC00130
ARCON
SMOVL C00131 BC00131 V=11.7  +MOVJ EC00131
ARCOF
SMOVL C00132 BC00132 V=800.0  +MOVJ EC00132
SMOVL C00133 BC00133 V=1000.0  +MOVJ EC00133
SFTOF3D
'EndPath W3431
'Path W3432
SFTOF3D
SFTON3D P030
MOVJ C00134 BC00134 VJ=100.00  +MOVJ EC00134 VJ=100.00
SMOVL C00135 BC00135 V=800.0  +MOVJ EC00135
SMOVL C00136 BC00136 V=150.0 PL=0  +MOVJ EC00136
MACRO1 MJ#(0) ARGF21
ARCON
SFTON3D P031
SMOVL C00137 BC00137 V=9.2  +MOVJ EC00137
ARCOF
SMOVL C00138 BC00138 V=800.0  +MOVJ EC00138
SMOVL C00139 BC00139 V=1000.0  +MOVJ EC00139
SFTOF3D
'EndPath W3432
'
MOVJ C00140 BC00140 VJ=100.00  +MOVJ EC00140 VJ=100.00
'
'Path W3434
SFTOF3D
SFTON3D P032
MOVJ C00141 BC00141 VJ=100.00  +MOVJ EC00141 VJ=100.00
SMOVL C00142 BC00142 V=800.0  +MOVJ EC00142
SMOVL C00143 BC00143 V=150.0 PL=0  +MOVJ EC00143
ARCON
SFTON3D P033
SMOVL C00144 BC00144 V=9.2  +MOVJ EC00144
SMOVL C00145 BC00145 V=9.2  +MOVJ EC00145
ARCOF
SMOVL C00146 BC00146 V=800.0  +MOVJ EC00146
SMOVL C00147 BC00147 V=1000.0  +MOVJ EC00147
SFTOF3D
'EndPath W3434
MOVJ C00148 BC00148 VJ=100.00  +MOVJ EC00148 VJ=100.00
'
MOVJ C00149 BC00149 VJ=100.00  +MOVJ EC00149 VJ=100.00
MOVJ C00150 BC00150 VJ=100.00  +MOVJ EC00150 VJ=100.00
MOVJ C00151 BC00151 VJ=100.00  +MOVJ EC00151 VJ=100.00
MOVJ C00152 BC00152 VJ=100.00  +MOVJ EC00152 VJ=100.00
MOVJ C00153 BC00153 VJ=100.00  +MOVJ EC00153 VJ=100.00
MOVJ C00154 BC00154 VJ=100.00  +MOVJ EC00154 VJ=100.00
CALL JOB:CLEAN-R1_KM_NEW
MOVJ C00155 BC00155 VJ=100.00  +MOVJ EC00155 VJ=100.00
MOVJ C00156 BC00156 VJ=100.00  +MOVJ EC00156 VJ=100.00
MOVJ C00157 BC00157 VJ=100.00  +MOVJ EC00157 VJ=100.00
MOVJ C00158 BC00158 VJ=100.00  +MOVJ EC00158 VJ=100.00
'
'Path S3435
SFTOF3D
MOVJ C00159 BC00159 VJ=100.00  +MOVJ EC00159 VJ=100.00
MOVL C00160 BC00160 V=666.7  +MOVJ EC00160 VJ=100.00
MOVL C00161 BC00161 V=666.7  +MOVJ EC00161 VJ=100.00
SMOVL C00162 BC00162 V=166.7  +MOVJ EC00162
SREFP 3 C00163 BC00163  +REFP EC00163
CALL JOB:SEARCH-R1-S13D
SET P041 P006
SFTON3D P041
SMOVL C00164 BC00164 V=166.7  +MOVJ EC00164
SREFP 3 C00165 BC00165  +REFP EC00165
CALL JOB:SEARCH-R1-S13D
SET P041 P006
SFTON3D P041
SMOVL C00166 BC00166 V=166.7  +MOVJ EC00166
MOVL C00167 BC00167 V=1000.0  +MOVJ EC00167 VJ=100.00
'EndPath S3435
'Path S3436
SFTOF3D
MOVJ C00168 BC00168 VJ=100.00  +MOVJ EC00168 VJ=100.00
MOVL C00169 BC00169 V=800.0  +MOVJ EC00169 VJ=100.00
SMOVL C00170 BC00170 V=166.7  +MOVJ EC00170
SREFP 3 C00171 BC00171  +REFP EC00171
CALL JOB:SEARCH-R1-S13D
SET P042 P006
SFTON3D P042
SMOVL C00172 BC00172 V=166.7  +MOVJ EC00172
SREFP 3 C00173 BC00173  +REFP EC00173
CALL JOB:SEARCH-R1-S13D
SET P042 P006
SFTON3D P042
SMOVL C00174 BC00174 V=166.7  +MOVJ EC00174
MOVL C00175 BC00175 V=1000.0  +MOVJ EC00175 VJ=100.00
'EndPath S3436
MOVJ C00176 BC00176 VJ=100.00  +MOVJ EC00176 VJ=100.00
MOVJ C00177 BC00177 VJ=100.00  +MOVJ EC00177 VJ=100.00
'Path S3438
SFTOF3D
MOVJ C00178 BC00178 VJ=100.00  +MOVJ EC00178 VJ=100.00
MOVL C00179 BC00179 V=800.0  +MOVJ EC00179 VJ=100.00
SMOVL C00180 BC00180 V=166.7  +MOVJ EC00180
SREFP 3 C00181 BC00181  +REFP EC00181
CALL JOB:SEARCH-R1-S13D
SET P044 P006
SFTON3D P044
SMOVL C00182 BC00182 V=166.7  +MOVJ EC00182
SREFP 3 C00183 BC00183  +REFP EC00183
CALL JOB:SEARCH-R1-S13D
SET P044 P006
SFTON3D P044
SMOVL C00184 BC00184 V=166.7  +MOVJ EC00184
MOVL C00185 BC00185 V=1000.0  +MOVJ EC00185 VJ=100.00
'EndPath S3438
'Path S3439
SFTOF3D
MOVJ C00186 BC00186 VJ=100.00  +MOVJ EC00186 VJ=100.00
MOVL C00187 BC00187 V=800.0  +MOVJ EC00187 VJ=100.00
SMOVL C00188 BC00188 V=166.7  +MOVJ EC00188
SREFP 3 C00189 BC00189  +REFP EC00189
CALL JOB:SEARCH-R1-S13D
SET P045 P006
SFTON3D P045
SMOVL C00190 BC00190 V=166.7  +MOVJ EC00190
SREFP 3 C00191 BC00191  +REFP EC00191
CALL JOB:SEARCH-R1-S13D
SET P045 P006
SFTON3D P045
SMOVL C00192 BC00192 V=166.7  +MOVJ EC00192
MOVL C00193 BC00193 V=1000.0  +MOVJ EC00193 VJ=100.00
'EndPath S3439
MOVJ C00194 BC00194 VJ=100.00  +MOVJ EC00194 VJ=100.00
'Path S3441
SFTOF3D
MOVJ C00195 BC00195 VJ=100.00  +MOVJ EC00195 VJ=100.00
MOVL C00196 BC00196 V=800.0  +MOVJ EC00196 VJ=100.00
SMOVL C00197 BC00197 V=166.7  +MOVJ EC00197
SREFP 3 C00198 BC00198  +REFP EC00198
CALL JOB:SEARCH-R1-S13D
SET P047 P006
SFTON3D P047
SMOVL C00199 BC00199 V=166.7  +MOVJ EC00199
SREFP 3 C00200 BC00200  +REFP EC00200
CALL JOB:SEARCH-R1-S13D
SET P047 P006
SFTON3D P047
SMOVL C00201 BC00201 V=166.7  +MOVJ EC00201
MOVL C00202 BC00202 V=1000.0  +MOVJ EC00202 VJ=100.00
'EndPath S3441
'Path S3442
SFTOF3D
MOVJ C00203 BC00203 VJ=100.00  +MOVJ EC00203 VJ=100.00
MOVL C00204 BC00204 V=800.0  +MOVJ EC00204 VJ=100.00
SMOVL C00205 BC00205 V=166.7  +MOVJ EC00205
SREFP 3 C00206 BC00206  +REFP EC00206
CALL JOB:SEARCH-R1-S13D
SET P048 P006
SFTON3D P048
SMOVL C00207 BC00207 V=166.7  +MOVJ EC00207
SREFP 3 C00208 BC00208  +REFP EC00208
CALL JOB:SEARCH-R1-S13D
SET P048 P006
SFTON3D P048
SMOVL C00209 BC00209 V=166.7  +MOVJ EC00209
MOVL C00210 BC00210 V=1000.0  +MOVJ EC00210 VJ=100.00
'EndPath S3442
'Path S3444
SFTOF3D
MOVJ C00211 BC00211 VJ=100.00  +MOVJ EC00211 VJ=100.00
MOVJ C00212 BC00212 VJ=100.00  +MOVJ EC00212 VJ=100.00
MOVL C00213 BC00213 V=800.0  +MOVJ EC00213 VJ=100.00
SMOVL C00214 BC00214 V=166.7  +MOVJ EC00214
SREFP 3 C00215 BC00215  +REFP EC00215
CALL JOB:SEARCH-R1-S13D
SET P050 P006
SFTON3D P050
SMOVL C00216 BC00216 V=166.7  +MOVJ EC00216
SREFP 3 C00217 BC00217  +REFP EC00217
CALL JOB:SEARCH-R1-S13D
SET P050 P006
SFTON3D P050
SMOVL C00218 BC00218 V=166.7  +MOVJ EC00218
MOVL C00219 BC00219 V=1000.0  +MOVJ EC00219 VJ=100.00
'EndPath S3444
'Path S3445
SFTOF3D
MOVJ C00220 BC00220 VJ=100.00  +MOVJ EC00220 VJ=100.00
MOVL C00221 BC00221 V=800.0  +MOVJ EC00221 VJ=100.00
SMOVL C00222 BC00222 V=166.7  +MOVJ EC00222
SREFP 3 C00223 BC00223  +REFP EC00223
CALL JOB:SEARCH-R1-S13D
SET P051 P006
SFTON3D P051
SMOVL C00224 BC00224 V=166.7  +MOVJ EC00224
SREFP 3 C00225 BC00225  +REFP EC00225
CALL JOB:SEARCH-R1-S13D
SET P051 P006
SFTON3D P051
SMOVL C00226 BC00226 V=166.7  +MOVJ EC00226
MOVL C00227 BC00227 V=1000.0  +MOVJ EC00227 VJ=100.00
'EndPath S3445
MOVJ C00228 BC00228 VJ=100.00  +MOVJ EC00228 VJ=100.00
'Path S3446
SFTOF3D
MOVJ C00229 BC00229 VJ=100.00  +MOVJ EC00229 VJ=100.00
MOVL C00230 BC00230 V=800.0  +MOVJ EC00230 VJ=100.00
SMOVL C00231 BC00231 V=166.7  +MOVJ EC00231
SREFP 3 C00232 BC00232  +REFP EC00232
CALL JOB:SEARCH-R1-S13D
SET P052 P006
SFTON3D P052
SMOVL C00233 BC00233 V=166.7  +MOVJ EC00233
SREFP 3 C00234 BC00234  +REFP EC00234
CALL JOB:SEARCH-R1-S13D
SET P052 P006
SFTON3D P052
SMOVL C00235 BC00235 V=166.7  +MOVJ EC00235
MOVL C00236 BC00236 V=1000.0  +MOVJ EC00236 VJ=100.00
'EndPath S3446
'Path S3447
SFTOF3D
MOVJ C00237 BC00237 VJ=100.00  +MOVJ EC00237 VJ=100.00
MOVL C00238 BC00238 V=800.0  +MOVJ EC00238 VJ=100.00
SMOVL C00239 BC00239 V=166.7  +MOVJ EC00239
SREFP 3 C00240 BC00240  +REFP EC00240
CALL JOB:SEARCH-R1-S13D
SET P053 P006
SFTON3D P053
SMOVL C00241 BC00241 V=166.7  +MOVJ EC00241
SREFP 3 C00242 BC00242  +REFP EC00242
CALL JOB:SEARCH-R1-S13D
SET P053 P006
SFTON3D P053
SMOVL C00243 BC00243 V=166.7  +MOVJ EC00243
MOVL C00244 BC00244 V=1000.0  +MOVJ EC00244 VJ=100.00
'EndPath S3447
'
'Path W3448
SFTOF3D
SFTON3D P052
MOVJ C00245 BC00245 VJ=100.00  +MOVJ EC00245 VJ=100.00
SMOVL C00246 BC00246 V=800.0  +MOVJ EC00246
SMOVL C00247 BC00247 V=150.0 PL=0  +MOVJ EC00247
ARCON
SFTON3D P053
SMOVL C00248 BC00248 V=9.2  +MOVJ EC00248
SMOVL C00249 BC00249 V=9.2  +MOVJ EC00249
ARCOF
SMOVL C00250 BC00250 V=800.0  +MOVJ EC00250
SMOVL C00251 BC00251 V=1000.0  +MOVJ EC00251
SFTOF3D
MOVJ C00252 BC00252 VJ=100.00  +MOVJ EC00252 VJ=100.00
'
'Path W3449
SFTOF3D
SFTON3D P050
MOVJ C00253 BC00253 VJ=100.00  +MOVJ EC00253 VJ=100.00
SMOVL C00254 BC00254 V=800.0  +MOVJ EC00254
SMOVL C00255 BC00255 V=150.0 PL=0  +MOVJ EC00255
ARCON
SFTON3D P051
SMOVL C00256 BC00256 V=9.2  +MOVJ EC00256
SMOVL C00257 BC00257 V=9.2  +MOVJ EC00257
ARCOF
SMOVL C00258 BC00258 V=800.0  +MOVJ EC00258
SMOVL C00259 BC00259 V=1000.0  +MOVJ EC00259
SFTOF3D
'EndPath W3449
'
'Path W3450
SFTOF3D
SFTON3D P047
MOVJ C00260 BC00260 VJ=100.00  +MOVJ EC00260 VJ=100.00
SMOVL C00261 BC00261 V=800.0  +MOVJ EC00261
'SPRAWDZONE DO TEGO PKT
SMOVL C00262 BC00262 V=150.0 PL=0  +MOVJ EC00262
MACRO1 MJ#(0) ARGF9
ARCON
SMOVL C00263 BC00263 V=11.7  +MOVJ EC00263
ARCOF
SMOVL C00264 BC00264 V=800.0  +MOVJ EC00264
SMOVL C00265 BC00265 V=1000.0  +MOVJ EC00265
SFTOF3D
'EndPath W3450
'Path W3451
SFTOF3D
SFTON3D P048
MOVJ C00266 BC00266 VJ=100.00  +MOVJ EC00266 VJ=100.00
SMOVL C00267 BC00267 V=800.0  +MOVJ EC00267
SMOVL C00268 BC00268 V=150.0 PL=0  +MOVJ EC00268
ARCON
SMOVL C00269 BC00269 V=11.7  +MOVJ EC00269
ARCOF
SMOVL C00270 BC00270 V=800.0  +MOVJ EC00270
SMOVL C00271 BC00271 V=1000.0  +MOVJ EC00271
SFTOF3D
'EndPath W3451
MOVJ C00272 BC00272 VJ=100.00  +MOVJ EC00272 VJ=100.00
'
'Path W3453
SFTOF3D
SFTON3D P044
MOVJ C00273 BC00273 VJ=100.00  +MOVJ EC00273 VJ=100.00
SMOVL C00274 BC00274 V=800.0  +MOVJ EC00274
SMOVL C00275 BC00275 V=150.0 PL=0  +MOVJ EC00275
ARCON
SMOVL C00276 BC00276 V=11.7  +MOVJ EC00276
ARCOF
SMOVL C00277 BC00277 V=800.0  +MOVJ EC00277
SMOVL C00278 BC00278 V=1000.0  +MOVJ EC00278
SFTOF3D
'EndPath W3453
'Path W3454
SFTOF3D
SFTON3D P045
MOVJ C00279 BC00279 VJ=100.00  +MOVJ EC00279 VJ=100.00
SMOVL C00280 BC00280 V=800.0  +MOVJ EC00280
SMOVL C00281 BC00281 V=150.0 PL=0  +MOVJ EC00281
ARCON
SMOVL C00282 BC00282 V=11.7  +MOVJ EC00282
ARCOF
SMOVL C00283 BC00283 V=800.0  +MOVJ EC00283
SMOVL C00284 BC00284 V=1000.0  +MOVJ EC00284
SFTOF3D
'EndPath W3454
MOVJ C00285 BC00285 VJ=100.00  +MOVJ EC00285 VJ=100.00
'
'
'Path W3456
SFTOF3D
SFTON3D P041
MOVJ C00286 BC00286 VJ=100.00  +MOVJ EC00286 VJ=100.00
SMOVL C00287 BC00287 V=800.0  +MOVJ EC00287
SMOVL C00288 BC00288 V=150.0 PL=0  +MOVJ EC00288
ARCON
SMOVL C00289 BC00289 V=11.7  +MOVJ EC00289
ARCOF
SMOVL C00290 BC00290 V=800.0  +MOVJ EC00290
SMOVL C00291 BC00291 V=1000.0  +MOVJ EC00291
SFTOF3D
'EndPath W3456
'Path W3457
SFTOF3D
SFTON3D P042
MOVJ C00292 BC00292 VJ=100.00  +MOVJ EC00292 VJ=100.00
SMOVL C00293 BC00293 V=800.0  +MOVJ EC00293
SMOVL C00294 BC00294 V=150.0 PL=0  +MOVJ EC00294
ARCON
SMOVL C00295 BC00295 V=11.7  +MOVJ EC00295
ARCOF
SMOVL C00296 BC00296 V=800.0  +MOVJ EC00296
SMOVL C00297 BC00297 V=1000.0  +MOVJ EC00297
SFTOF3D
'EndPath W3457
MOVJ C00298 BC00298 VJ=100.00  +MOVJ EC00298 VJ=100.00
MOVJ C00299 BC00299 VJ=100.00  +MOVJ EC00299 VJ=100.00
MOVJ C00300 BC00300 VJ=100.00  +MOVJ EC00300 VJ=100.00
END
